# EPICS autosave request: GalilSup/Db/GALIL_settings.req
file "GALIL_controller_settings.req" P=$(P),CCP=01
file "GALIL_controller_settings.req" P=$(P),CCP=02
file "GALIL_controller_settings.req" P=$(P),CCP=03
file "GALIL_controller_settings.req" P=$(P),CCP=04
file "GALIL_controller_settings.req" P=$(P),CCP=05
file "GALIL_controller_settings.req" P=$(P),CCP=06
file "GALIL_controller_settings.req" P=$(P),CCP=07
